{attribute addProperty BoxType "AT2040-0250-0021"}
{attribute addProperty Id "A_0108_AT2000_5233_0019_AT2000_5233AT2000_C5E5984862678.25"}
{attribute addProperty CRC "2743623356"}
{attribute addProperty SizeInBites "626"}
{attribute addProperty SizeInBytes "78.25"}
TYPE A_0036_AT2040_0250_0021_A3885EBC EXTENDS AT2040_BA5A9548 :
STRUCT
	{attribute addProperty Name "A_0108_AT2000_5233_0019_AT2000_5233"}
	A_0108_AT2000_5233_0019_AT2000_5233 : AT2000_C5E59848;
END_STRUCT
END_TYPE

(* stored: Version 1.2.0.0, ProductVersion 3.1.4024.9
   DUT A_0036_AT2040_0250_0021_A3885EBC: Id {dec5e5ba-405e-4406-bbb0-be6feafe43ea} *)
